Staubli VAL3: CartesianForce.dtx

public num cf[6]
public num resForce
